# EPICS autosave request: leybold/read_write_int_settings.req
$(P):$(PARAM)
